# EPICS substitutions: iocBoot/ioc13LQExcel/asynRecord.substitutions
file "$(ASYN)/db/asynRecord.db"
{
pattern
{P              R         PORT     ADDR  OMAX IMAX}
{13LQE1:       serial1   serial1    0    256  256}
}
